{attribute 'qualified_only'}
{attribute 'strict'}
{attribute 'to_string'}
TYPE E_3002_Status : (
		Not_ok := 0, //ERROR_PLC_FAILURE will be activated, and additionally manual driving will be prevented.
		Ok	   := 1	 //Navitrol is allowed to drive the AGV.
	) UINT;
END_TYPE

(* stored: Version 1.1.0.1, ProductVersion 3.1.4026.17
   DUT E_3002_Status: Id {6b4550bd-3809-4ca2-b45c-62dd3266659a} *)
